FUNCTION_BLOCK ENCODER2ANGLE
VAR_INPUT
	enc_a : BOOL;
	enc_b : BOOL;
END_VAR
VAR_OUTPUT
	enc_pulsecount : DINT;
	enc_angle : REAL;
END_VAR
VAR
END_VAR

END_FUNCTION_BLOCK

(* stored: Version 1.1.0.1, ProductVersion 3.1.4024.4
   POU ENCODER2ANGLE: Id {8f1b6799-8175-42cd-a06b-61058091be48}, SpecialFunc None *)
